(*

.. <legal notes>

legal notes
=================
| SPDX-FileCopyrightText: © 2026 Oleksandr Tiutyk <trofimich@gmail.com>
| SPDX-License-Identifier: LGPL-3.0-only
| For details check: LGPL-3.0-only_

.. _LGPL-3.0-only: https://www.gnu.org/licenses/lgpl-3.0.en.html

.. </legal notes>

*)

{attribute 'no_explicit_call' := 'do not call this function block directly'} 
PROGRAM Terminals
VAR_OUTPUT
	DI_1 : TOF_IOModels.EL1018;
	DO_2 : TOF_IOModels.EL2409;
	AI_3 : TOF_IOModels.EL3001;
END_VAR

END_PROGRAM

(* stored: Version 1.1.0.1
   POU Terminals: Id {a98d253d-f32d-4c19-9c5a-20b1f705b795}, SpecialFunc None *)
